(* PLC project SafeLOGIC-1, BrAutomation SafeDESIGNER  4.3.2.11 *)
(* stored: companyURL http://www.br-automation.com, creationDateTime Tue Mar 06 09:32:48 2018 *)

PROGRAM Main

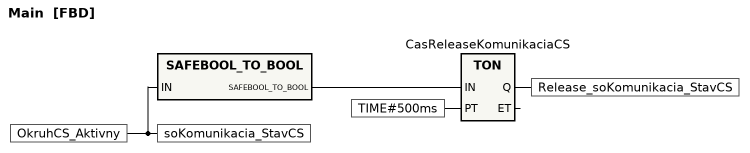
(* FBD diagram, written out as Structured Text *)
soKomunikacia_StavCS := OkruhCS_Aktivny;
CasReleaseKomunikaciaCS(IN := SAFEBOOL_TO_BOOL(OkruhCS_Aktivny), PT := TIME#500ms);
Release_soKomunikacia_StavCS := CasReleaseKomunikaciaCS.Q;
END_PROGRAM
